PROGRAM MAIN
VAR
END_VAR

END_PROGRAM

(* stored: Version 1.1.0.1
   POU MAIN: Id {3eab0344-5321-42e5-b1b4-0c216c60fbfd} *)
